// TIA Portal project "bai_lam_phan_loai_sp_qr_code" (V16)

(* hardware
DEVICE "S7-1200 station_1"  S7-1200 Station
   slot 0: "Rack_0"  S7-1200 Rack  Rack  V1.0
   slot 1: "PLC_1"  CPU 1214C DC/DC/DC  6ES7 214-1AG40-0XB0  V4.4
DEVICE "PC-System_1"  SIMATIC PC station
   slot 0: "SIMATIC PC station"  Rail  SIMATIC PC-Station  V1.0
      slot 125: "Stationmanager"  Station_Manager  V6.0.4
   slot 1: "HMI_RT_1"  WinCC RT Advanced  6AV2 104-0xxxx-xxxx  16.0.0.0
      slot 33792: "Computer interface"  Host interface
   slot 2: "IE general_1"  IE General  IE_CP  V8.2.0
*)

// ===== PLC "PLC_1"  CPU 1214C DC/DC/DC =====

VAR_GLOBAL   // PLC tag table "Auto"
   "START" AT %I0.0 : Bool;
   "STOP" AT %I0.1 : Bool;
   "CB_phat_hien" AT %I0.2 : Bool;
   "CB_XILANH1" AT %I0.3 : Bool;
   "CB_XILANH2" AT %I0.4 : Bool;
   "CB_XILANH3" AT %I0.5 : Bool;
   "CB_XILANH4" AT %I0.6 : Bool;
   "CB_XILANH5" AT %I0.7 : Bool;
   "BANGTAI" AT %Q0.0 : Bool;
   "XILANH1" AT %Q0.1 : Bool;
   "XILANH2" AT %Q0.2 : Bool;
   "XILANH3" AT %Q0.3 : Bool;
   "XILANH4" AT %Q0.4 : Bool;
   "XILANH5" AT %Q0.5 : Bool;
   "Den_bao_day" AT %Q0.6 : Bool;
   "Q_AUTO" AT %M1.0 : Bool;
   "duy_tri" AT %M1.1 : Bool;
   "bien_nho1" AT %M1.2 : Bool;
   "bien_nho2" AT %M1.3 : Bool;
   "bien_nho3" AT %M1.4 : Bool;
   "bien_nho4" AT %M1.5 : Bool;
   "bien_nho5" AT %M1.6 : Bool;
   "value_ofkey" AT %MW20 : Int;
   "Detect_press" AT %M3.0 : Bool;
   "delay_2s" AT %M3.1 : Bool;
END_VAR

VAR_GLOBAL   // PLC tag table "MANU"
   "M_MANU_BANGTAI" AT %M0.0 : Bool;
   "M_XILANH1_MANU" AT %M0.1 : Bool;
   "M_XILANH2_MANU" AT %M0.2 : Bool;
   "M_XILANH3_MANU" AT %M0.3 : Bool;
   "M_XILANH4_MANU" AT %M0.4 : Bool;
   "M_XILANH5_MANU" AT %M0.5 : Bool;
   "Q_MANU" AT %M0.6 : Bool;
END_VAR

DATA_BLOCK "Data_Python"   // DB1
{ S7_Optimized_Access := 'TRUE' }
VERSION : 0.1
   VAR
      DBX_QR : Array[0..0] of Int;
      DBX_MA1 : Bool;
      DBX_MA2 : Bool;
      DBX_MA3 : Bool;
      DBX_MA4 : Bool;
      DBX_MA5 : Bool;
   END_VAR
BEGIN
END_DATA_BLOCK

DATA_BLOCK "Data_Move_BLk"   // DB2
{ S7_Optimized_Access := 'TRUE' }
VERSION : 0.1
   VAR
      Source : Array[0..0] of Int;
      Dest : Array[1..5] of Int;
      Count : UDInt;
      Source_index : Int;
      Dest_index : Int;
      "Return" : Int;
      Out_Buff : Array[0..0] of Int;
   END_VAR
BEGIN
END_DATA_BLOCK

// folder: System blocks/Program resources

DATA_BLOCK "T1"   // DB3
{ S7_Optimized_Access := 'TRUE' }
AUTHOR : Simatic
FAMILY : IEC
NAME : CNTR
VERSION : 1.0
// stored: InstanceOfName IEC_COUNTER
"IEC_COUNTER"
BEGIN
END_DATA_BLOCK

DATA_BLOCK "T2"   // DB4
{ S7_Optimized_Access := 'TRUE' }
AUTHOR : Simatic
FAMILY : IEC
NAME : IEC_TMR
VERSION : 1.0
// stored: InstanceOfName IEC_TIMER
"IEC_TIMER"
BEGIN
END_DATA_BLOCK

DATA_BLOCK "T3"   // DB5
{ S7_Optimized_Access := 'TRUE' }
AUTHOR : Simatic
FAMILY : IEC
NAME : CNTR
VERSION : 1.0
// stored: InstanceOfName IEC_COUNTER
"IEC_COUNTER"
BEGIN
END_DATA_BLOCK

DATA_BLOCK "T4"   // DB6
{ S7_Optimized_Access := 'TRUE' }
AUTHOR : Simatic
FAMILY : IEC
NAME : CNTR
VERSION : 1.0
// stored: InstanceOfName IEC_COUNTER
"IEC_COUNTER"
BEGIN
END_DATA_BLOCK

// folder: (top level)

FUNCTION "Auto" : Void   // FC1, LAD
{ S7_Optimized_Access := 'TRUE' }
VERSION : 0.1
   VAR_TEMP   // added for the SCL form of the ladder/FBD networks
      _w1 : Bool;
      _w2 : Bool;
      _w3 : Bool;
      _w4 : Bool;
      _w5 : Bool;
      _w6 : Bool;
   END_VAR
BEGIN

REGION Network 1: khởi động băng tải và đếm sản phẩm vào
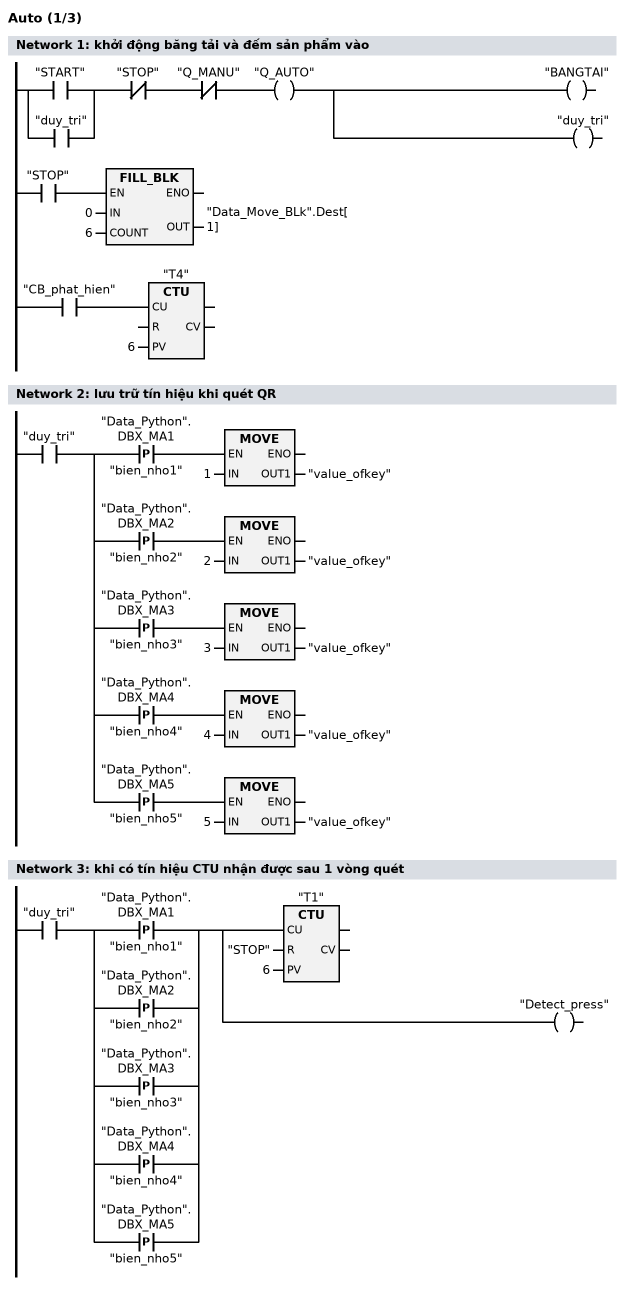
   "Q_AUTO" := ("START" OR "duy_tri") AND NOT "STOP" AND NOT "Q_MANU";
   "BANGTAI" := "Q_AUTO";
   "duy_tri" := "Q_AUTO";
   IF "STOP" THEN FILL_BLK(IN := 0, COUNT := 6, OUT => "Data_Move_BLk".Dest[1]); END_IF;
   "T4".CTU(CU := "CB_phat_hien", PV := 6);
END_REGION

REGION Network 2: lưu trữ tín hiệu khi quét QR
   RUNG wire#powerrail
      Contact( "duy_tri" )
      wire#w1
      P_Contact(operand := "Data_Python".DBX_MA1, bit := "bien_nho1")
      Move(in := 1, out1 => "value_ofkey")
   END_RUNG
   RUNG wire#w1
      P_Contact(operand := "Data_Python".DBX_MA2, bit := "bien_nho2")
      Move(in := 2, out1 => "value_ofkey")
   END_RUNG
   RUNG wire#w1
      P_Contact(operand := "Data_Python".DBX_MA3, bit := "bien_nho3")
      Move(in := 3, out1 => "value_ofkey")
   END_RUNG
   RUNG wire#w1
      P_Contact(operand := "Data_Python".DBX_MA4, bit := "bien_nho4")
      Move(in := 4, out1 => "value_ofkey")
   END_RUNG
   RUNG wire#w1
      P_Contact(operand := "Data_Python".DBX_MA5, bit := "bien_nho5")
      Move(in := 5, out1 => "value_ofkey")
   END_RUNG
   // the same network as SCL:
   #_w1 := "duy_tri" AND "Data_Python".DBX_MA1 AND NOT "bien_nho1";   // rising edge of "Data_Python".DBX_MA1
   "bien_nho1" := "Data_Python".DBX_MA1;
   IF #_w1 THEN "value_ofkey" := 1; END_IF;
   #_w2 := "duy_tri" AND "Data_Python".DBX_MA2 AND NOT "bien_nho2";   // rising edge of "Data_Python".DBX_MA2
   "bien_nho2" := "Data_Python".DBX_MA2;
   IF #_w2 THEN "value_ofkey" := 2; END_IF;
   #_w3 := "duy_tri" AND "Data_Python".DBX_MA3 AND NOT "bien_nho3";   // rising edge of "Data_Python".DBX_MA3
   "bien_nho3" := "Data_Python".DBX_MA3;
   IF #_w3 THEN "value_ofkey" := 3; END_IF;
   #_w4 := "duy_tri" AND "Data_Python".DBX_MA4 AND NOT "bien_nho4";   // rising edge of "Data_Python".DBX_MA4
   "bien_nho4" := "Data_Python".DBX_MA4;
   IF #_w4 THEN "value_ofkey" := 4; END_IF;
   #_w5 := "duy_tri" AND "Data_Python".DBX_MA5 AND NOT "bien_nho5";   // rising edge of "Data_Python".DBX_MA5
   "bien_nho5" := "Data_Python".DBX_MA5;
   IF #_w5 THEN "value_ofkey" := 5; END_IF;
END_REGION

REGION Network 3: khi có tín hiệu CTU nhận được sau 1 vòng quét
   #_w1 := "duy_tri" AND "Data_Python".DBX_MA1 AND NOT "bien_nho1";   // rising edge of "Data_Python".DBX_MA1
   "bien_nho1" := "Data_Python".DBX_MA1;
   #_w2 := "duy_tri" AND "Data_Python".DBX_MA2 AND NOT "bien_nho2";   // rising edge of "Data_Python".DBX_MA2
   "bien_nho2" := "Data_Python".DBX_MA2;
   #_w3 := "duy_tri" AND "Data_Python".DBX_MA3 AND NOT "bien_nho3";   // rising edge of "Data_Python".DBX_MA3
   "bien_nho3" := "Data_Python".DBX_MA3;
   #_w4 := "duy_tri" AND "Data_Python".DBX_MA4 AND NOT "bien_nho4";   // rising edge of "Data_Python".DBX_MA4
   "bien_nho4" := "Data_Python".DBX_MA4;
   #_w5 := "duy_tri" AND "Data_Python".DBX_MA5 AND NOT "bien_nho5";   // rising edge of "Data_Python".DBX_MA5
   "bien_nho5" := "Data_Python".DBX_MA5;
   #_w6 := #_w1 OR #_w2 OR #_w3 OR #_w4 OR #_w5;
   "T1".CTU(CU := #_w6, R := "STOP", PV := 6);
   "Detect_press" := #_w6;
END_REGION

REGION Network 4: chuyển dần các giá trị dần vào hàm để nhớ
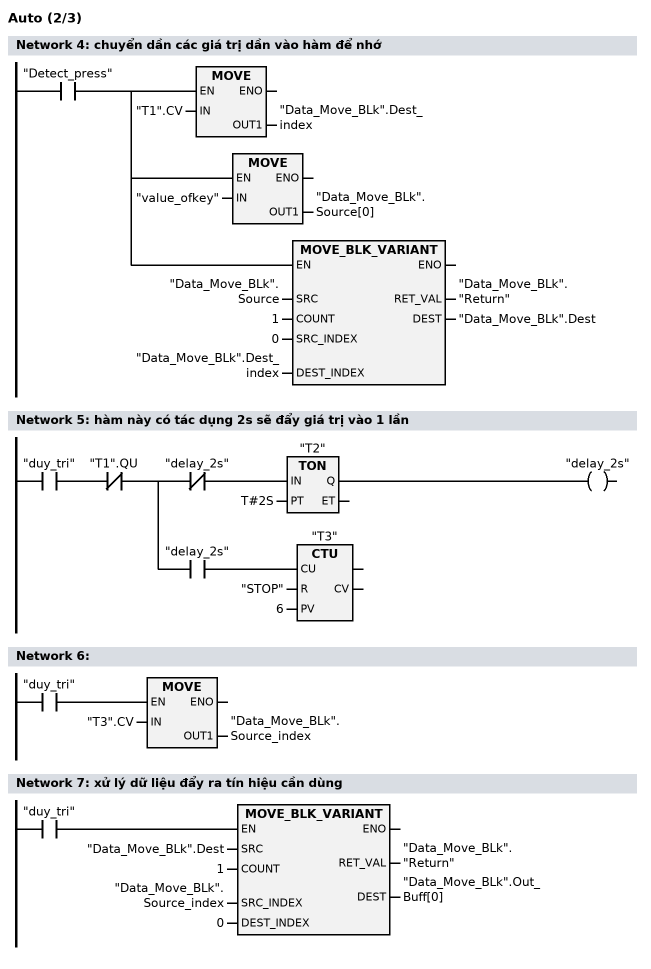
   IF "Detect_press" THEN
       "Data_Move_BLk".Dest_index := "T1".CV;
       "Data_Move_BLk".Source[0] := "value_ofkey";
       "Data_Move_BLk"."Return" := MOVE_BLK_VARIANT(SRC := "Data_Move_BLk".Source,
                               COUNT := 1,
                               SRC_INDEX := 0,
                               DEST_INDEX := "Data_Move_BLk".Dest_index,
                               DEST => "Data_Move_BLk".Dest);
   END_IF;
END_REGION

REGION Network 5: hàm này có tác dụng 2s sẽ đẩy giá trị vào 1 lần
   #_w1 := "duy_tri" AND NOT "T1".QU;
   "T2".TON(IN := #_w1 AND NOT "delay_2s", PT := T#2S);
   "delay_2s" := "T2".Q;
   "T3".CTU(CU := #_w1 AND "delay_2s", R := "STOP", PV := 6);
END_REGION

REGION Network 6
   RUNG wire#powerrail
      Contact( "duy_tri" )
      Move(in := "T3".CV, out1 => "Data_Move_BLk".Source_index)
   END_RUNG
   // the same network as SCL:
   IF "duy_tri" THEN "Data_Move_BLk".Source_index := "T3".CV; END_IF;
END_REGION

REGION Network 7: xử lý dữ liệu đẩy ra tín hiệu cần dùng
   IF "duy_tri" THEN
       "Data_Move_BLk"."Return" := MOVE_BLK_VARIANT(SRC := "Data_Move_BLk".Dest,
                               COUNT := 1,
                               SRC_INDEX := "Data_Move_BLk".Source_index,
                               DEST_INDEX := 0,
                               DEST => "Data_Move_BLk".Out_Buff[0]);
   END_IF;
END_REGION

REGION Network 8: tín hiệu được đẩy ra theo thứ tự tín hiệu gửi về
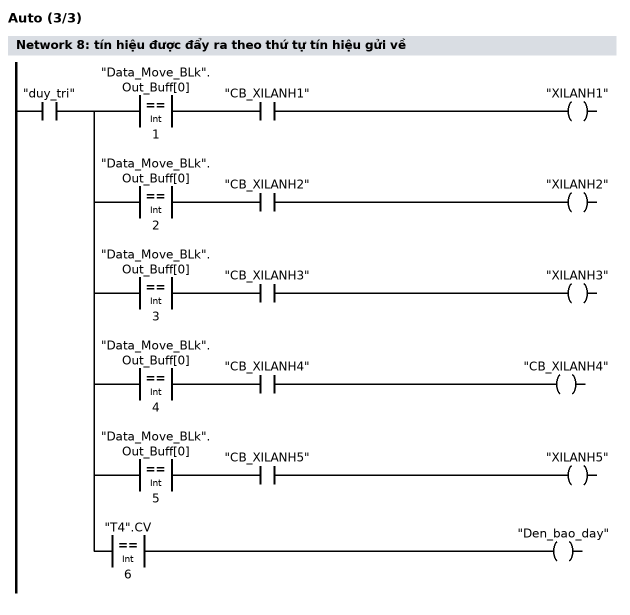
   RUNG wire#powerrail
      Contact( "duy_tri" )
      wire#w1
      { S7_Templates := "SrcType := Int" } EQ_Contact(in1 := "Data_Move_BLk".Out_Buff[0], in2 := 1)
      Contact( "CB_XILANH1" )
      Coil( "XILANH1" )
   END_RUNG
   RUNG wire#w1
      { S7_Templates := "SrcType := Int" } EQ_Contact(in1 := "Data_Move_BLk".Out_Buff[0], in2 := 2)
      Contact( "CB_XILANH2" )
      Coil( "XILANH2" )
   END_RUNG
   RUNG wire#w1
      { S7_Templates := "SrcType := Int" } EQ_Contact(in1 := "Data_Move_BLk".Out_Buff[0], in2 := 3)
      Contact( "CB_XILANH3" )
      Coil( "XILANH3" )
   END_RUNG
   RUNG wire#w1
      { S7_Templates := "SrcType := Int" } EQ_Contact(in1 := "Data_Move_BLk".Out_Buff[0], in2 := 4)
      Contact( "CB_XILANH4" )
      Coil( "CB_XILANH4" )
   END_RUNG
   RUNG wire#w1
      { S7_Templates := "SrcType := Int" } EQ_Contact(in1 := "Data_Move_BLk".Out_Buff[0], in2 := 5)
      Contact( "CB_XILANH5" )
      Coil( "XILANH5" )
   END_RUNG
   RUNG wire#w1
      { S7_Templates := "SrcType := Int" } EQ_Contact(in1 := "T4".CV, in2 := 6)
      Coil( "Den_bao_day" )
   END_RUNG
   // the same network as SCL:
   "XILANH1" := "duy_tri" AND ("Data_Move_BLk".Out_Buff[0] = 1) AND "CB_XILANH1";
   "XILANH2" := "duy_tri" AND ("Data_Move_BLk".Out_Buff[0] = 2) AND "CB_XILANH2";
   "XILANH3" := "duy_tri" AND ("Data_Move_BLk".Out_Buff[0] = 3) AND "CB_XILANH3";
   "CB_XILANH4" := "duy_tri" AND ("Data_Move_BLk".Out_Buff[0] = 4) AND "CB_XILANH4";
   "XILANH5" := "duy_tri" AND ("Data_Move_BLk".Out_Buff[0] = 5) AND "CB_XILANH5";
   "Den_bao_day" := "duy_tri" AND ("T4".CV = 6);
END_REGION
END_FUNCTION

FUNCTION "Che_do_bang_tay" : Void   // FC2, LAD
{ S7_Optimized_Access := 'TRUE' }
VERSION : 0.1
BEGIN

REGION Network 1: chế độ bằng tay của băng tải
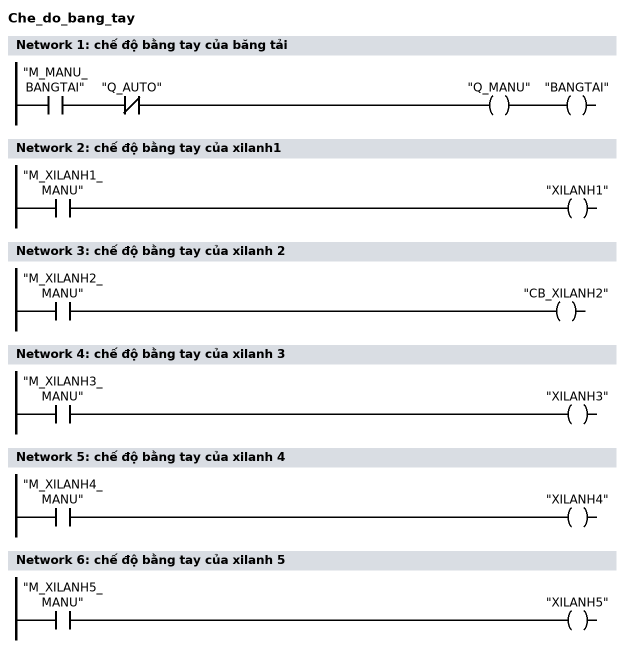
   RUNG wire#powerrail
      Contact( "M_MANU_BANGTAI" )
      I_Contact( "Q_AUTO" )
      Coil( "Q_MANU" )
      Coil( "BANGTAI" )
   END_RUNG
   // the same network as SCL:
   "Q_MANU" := "M_MANU_BANGTAI" AND NOT "Q_AUTO";
   "BANGTAI" := "Q_MANU";
END_REGION

REGION Network 2: chế độ bằng tay của xilanh1
   RUNG wire#powerrail
      Contact( "M_XILANH1_MANU" )
      Coil( "XILANH1" )
   END_RUNG
   // the same network as SCL:
   "XILANH1" := "M_XILANH1_MANU";
END_REGION

REGION Network 3: chế độ bằng tay của xilanh 2
   RUNG wire#powerrail
      Contact( "M_XILANH2_MANU" )
      Coil( "CB_XILANH2" )
   END_RUNG
   // the same network as SCL:
   "CB_XILANH2" := "M_XILANH2_MANU";
END_REGION

REGION Network 4: chế độ bằng tay của xilanh 3
   RUNG wire#powerrail
      Contact( "M_XILANH3_MANU" )
      Coil( "XILANH3" )
   END_RUNG
   // the same network as SCL:
   "XILANH3" := "M_XILANH3_MANU";
END_REGION

REGION Network 5: chế độ bằng tay của xilanh 4
   RUNG wire#powerrail
      Contact( "M_XILANH4_MANU" )
      Coil( "XILANH4" )
   END_RUNG
   // the same network as SCL:
   "XILANH4" := "M_XILANH4_MANU";
END_REGION

REGION Network 6: chế độ bằng tay của xilanh 5
   RUNG wire#powerrail
      Contact( "M_XILANH5_MANU" )
      Coil( "XILANH5" )
   END_RUNG
   // the same network as SCL:
   "XILANH5" := "M_XILANH5_MANU";
END_REGION
END_FUNCTION

ORGANIZATION_BLOCK "Main"   // OB1, LAD, ProgramCycle
TITLE = "Main Program Sweep (Cycle)"
{ S7_Optimized_Access := 'TRUE' }
VERSION : 0.1
   VAR_INPUT
      Initial_Call : Bool;   // Initial call of this OB
      Remanence : Bool;   // =True, if remanent data are available
   END_VAR
BEGIN

REGION Network 1: chế độ auto
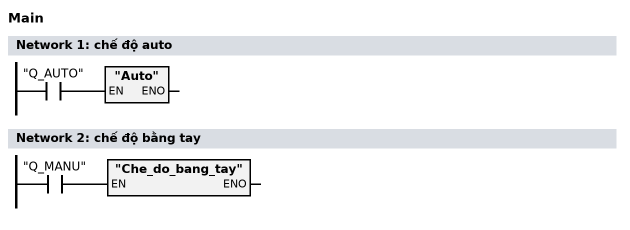
   RUNG wire#powerrail
      Contact( "Q_AUTO" )
      "Auto"()
   END_RUNG
   // the same network as SCL:
   IF "Q_AUTO" THEN "Auto"(); END_IF;
END_REGION

REGION Network 2: chế độ bằng tay
   RUNG wire#powerrail
      Contact( "Q_MANU" )
      "Che_do_bang_tay"()
   END_RUNG
   // the same network as SCL:
   IF "Q_MANU" THEN "Che_do_bang_tay"(); END_IF;
END_REGION
END_ORGANIZATION_BLOCK

(* ===== HMI "HMI_RT_1" =====
connection "HMI_Connection_1": ETHERNET, S7_1200_OMS

screen "Thiet_ke_giao_dien" 1024x768
   SymbolLibrary "Symbol library_1" at 34,470 size 315x45
   SymbolLibrary "Symbol library_3" at 274,470 size 301x45
   SymbolLibrary "Symbol library_2" at 422,470 size 315x45
   SymbolLibrary "Symbol library_4" at 554,470 size 315x45
   SymbolLibrary "Symbol library_5" at 613,470 size 370x44
   Group "Group_2" at 297,214 size 89x216
   SymbolLibrary "Symbol library_6" at 266,384 size 21x46
   SymbolLibrary "Symbol library_7" at 180,384 size 21x46
   Group "Group_5" at 433,214 size 89x216
   SymbolLibrary "Symbol library_8" at 402,384 size 21x46
   Group "Group_8" at 569,214 size 89x216
   SymbolLibrary "Symbol library_9" at 538,384 size 21x46
   Group "Group_11" at 705,214 size 89x216
   SymbolLibrary "Symbol library_10" at 674,384 size 21x46
   Group "Group_14" at 841,214 size 89x216
   SymbolLibrary "Symbol library_11" at 810,384 size 21x46
   TextField "Text field_1" at 104,357 size 127x20; Text 'cảm biến phát hiện'
   TextField "Text field_2" at 256,362 size 35x22; Text 'CB1'
   TextField "Text field_3" at 401,360 size 35x22; Text 'CB2'
   TextField "Text field_4" at 522,358 size 35x22; Text 'CB3'
   TextField "Text field_5" at 667,360 size 35x22; Text 'CB4'
   TextField "Text field_6" at 806,359 size 35x22; Text 'CB5'
   Switch "Switch_1" at 264,225 size 63x41; CaptionText 'Switch'; TextOff 'OFF'; TextOn 'ON'
   Switch "Switch_2" at 412,227 size 63x41; TextOn 'ON'; CaptionText 'Switch'; TextOff 'OFF'
   Switch "Switch_3" at 538,225 size 63x41; TextOn 'ON'; CaptionText 'Switch'; TextOff 'OFF'
   Switch "Switch_4" at 676,227 size 63x41; TextOn 'ON'; CaptionText 'Switch'; TextOff 'OFF'
   Switch "Switch_5" at 824,225 size 63x41; TextOn 'ON'; CaptionText 'Switch'; TextOff 'OFF'
   Group "Group_15" at 157,504 size 156x238
   Group "Group_16" at 291,504 size 156x238
   Group "Group_17" at 425,504 size 156x238
   Group "Group_18" at 559,504 size 156x238
   Group "Group_19" at 693,504 size 156x238
   Switch "Switch_6" at 27,42 size 184x88; CaptionText 'CHE DO VAN HANH'; TextOff 'MANU'; TextOn 'AUTO'
   Button "Button_1" at 23,150 size 96x32; TextOff 'START'
   Button "Button_2" at 140,150 size 96x32; TextOff 'STOP'
   Switch "Switch_7" at 72,610 size 63x41; TextOn 'ON'; CaptionText 'Switch'; TextOff 'OFF'
   TextField "Text field_7" at 322,55 size 47x22; Text 'AUTO'
   TextField "Text field_8" at 322,142 size 51x22; Text 'MANU'
   SymbolLibrary "Symbol library_17" at 52,522 size 120x79
   Group "Group" at 326,214 size 60x124
   Group "Group_1" at 297,321 size 56x109
   Group "Group_3" at 462,214 size 60x124
   Group "Group_4" at 433,321 size 56x109
   Group "Group_6" at 598,214 size 60x124
   Group "Group_7" at 569,321 size 56x109
   Group "Group_9" at 734,214 size 60x124
   Group "Group_10" at 705,321 size 56x109
   Group "Group_12" at 870,214 size 60x124
   Group "Group_13" at 841,321 size 56x109
   SymbolLibrary "Symbol library_12" at 157,665 size 155x77
   SymbolLibrary "Symbol library_13" at 291,665 size 155x77
   SymbolLibrary "Symbol library_14" at 425,665 size 155x77
   SymbolLibrary "Symbol library_15" at 559,665 size 155x77
   SymbolLibrary "Symbol library_16" at 693,665 size 155x77
*)